// TIA Portal V19 export
TYPE "dtStageDown"
   STRUCT
      zoneChangeOP { S7_SetPoint := 'True'} : Real := 40.0;
      prevOP { S7_SetPoint := 'True'} : Real := 20.0;
      nextOP { S7_SetPoint := 'True'} : Real := 70.0;
      stabilizeDelay { S7_SetPoint := 'True'} : Time := T#5s;
      followUp : Bool;
   END_STRUCT;
END_TYPE
